// TIA Portal V20 export
TYPE "typeEmAddedWorksPara"
// stored: Access Published, Namespace Unit1
   STRUCT
      "Bool" { S7_SetPoint := 'True'} : Array[0..200] of Bool;
      P_Pulse { S7_SetPoint := 'True'} : Array[0..50] of Bool;
      N_Pulse { S7_SetPoint := 'True'} : Array[0..50] of Bool;
      "Dint" { S7_SetPoint := 'True'} : Array[0..100] of DInt;
      Lreal { S7_SetPoint := 'True'} : Array[0..100] of LReal;
      "Time" { S7_SetPoint := 'True'} : Array[0..100] of IEC_TIMER;
      "String" { S7_SetPoint := 'True'} : Array[0..10] of String;
   END_STRUCT;
END_TYPE
